(* PLC project mtcs_tmc, Institute of Astronomy Onto 0.0.1 *)
(* stored: creationDateTime 2025-05-06T14:59:44.773808, modificationDateTime 2025-05-06T14:59:44.773808 *)

TYPE TmcTimingMode : (LOCAL_CLOCK := 0, PTP_IEEE_1588 := 1);
END_TYPE

TYPE TmcAxesErrors : (AXES_NO_ERROR := 0, AXES_OBJECT_RC_OUT_OF_RANGE := 1, AXES_OBJECT_DC_OUT_OF_RANGE := 2, AXES_OBJECT_PR_OUT_OF_RANGE := 3, AXES_OBJECT_PD_OUT_OF_RANGE := 4, AXES_OBJECT_PX_OUT_OF_RANGE := 5, AXES_EQ_OUT_OF_RANGE := 6, AXES_LOCATION_XP_OUT_OF_RANGE := 7, AXES_LOCATION_YP_OUT_OF_RANGE := 8, AXES_LOCATION_DX_OUT_OF_RANGE := 9, AXES_LOCATION_DY_OUT_OF_RANGE := 10, AXES_LOCATION_ELONG_OUT_OF_RANGE := 11, AXES_LOCATION_PHI_OUT_OF_RANGE := 12, AXES_LOCATION_HM_OUT_OF_RANGE := 13, AXES_LOCATION_TK_OUT_OF_RANGE := 14, AXES_LOCATION_PHPA_OUT_OF_RANGE := 15, AXES_LOCATION_RH_OUT_OF_RANGE := 16, AXES_LOCATION_WLFQ_OUT_OF_RANGE := 17, AXES_LOCATION_TLR_OUT_OF_RANGE := 18, AXES_FEEDBACK_AZ_OUT_OF_RANGE := 19, AXES_FEEDBACK_EL_OUT_OF_RANGE := 20);
END_TYPE

TYPE TmcTimingErrors : (TIMING_NO_ERROR := 0, TIMING_DUT_OUT_OF_RANGE := 1, TIMING_GETCURDCTIME_FAILED := 2);
END_TYPE

TYPE TmcTarget : STRUCT
  {attribute 'TcHmiSymbol.Show'}
  rc : LREAL;  (* Object mean right ascention (alpha) in radians *)
  {attribute 'TcHmiSymbol.Show'}
  dc : LREAL;  (* Object mean declination (delta) in radians *)
  {attribute 'TcHmiSymbol.Show'}
  pr : INT;  (* Object Right Ascention proper motion in radians/year (do not multiply by cos(dc)!) *)
  {attribute 'TcHmiSymbol.Show'}
  pd : INT;  (* Object declination proper motion in radians/year *)
  {attribute 'TcHmiSymbol.Show'}
  px : LREAL;  (* Object parallax in arcseconds *)
  {attribute 'TcHmiSymbol.Show'}
  rv : LREAL;  (* Object radial velocity in km/s *)
END_STRUCT;
END_TYPE

TYPE TmcLocation : STRUCT
  {attribute 'TcHmiSymbol.Show'}
  xp : REAL;  (* Earth polar motion x in radians *)
  {attribute 'TcHmiSymbol.Show'}
  yp : REAL;  (* Earth polar motion y in radians *)
  {attribute 'TcHmiSymbol.Show'}
  dx : REAL;  (* Nutation adjustment dX in radians *)
  {attribute 'TcHmiSymbol.Show'}
  dy : REAL;  (* Nutation adjustment dY in radians *)
  {attribute 'TcHmiSymbol.Show'}
  elong : LREAL;  (* East longitude in radians *)
  {attribute 'TcHmiSymbol.Show'}
  phi : LREAL;  (* latitude in radians *)
  {attribute 'TcHmiSymbol.Show'}
  hm : REAL;  (* Height above sea level in meters *)
  {attribute 'TcHmiSymbol.Show'}
  tk : REAL;  (* Local temperature in Kelvin *)
  {attribute 'TcHmiSymbol.Show'}
  phpa : REAL;  (* Local pressure in hectoPascal = millibar *)
  {attribute 'TcHmiSymbol.Show'}
  rh : REAL;  (* Local relative humidity as a fraction (0...1) *)
  {attribute 'TcHmiSymbol.Show'}
  wlfq : REAL;  (* Observing wavelength in microns *)
  {attribute 'TcHmiSymbol.Show'}
  tlr : REAL;  (* Tropospheric lapse rate in K/m *)
END_STRUCT;
END_TYPE

TYPE TmcAzEl : STRUCT
  {attribute 'TcHmiSymbol.Show'}
  az : LREAL;  (* Azimuth in radians *)
  {attribute 'TcHmiSymbol.Show'}
  el : LREAL;  (* Elevation in radians *)
END_STRUCT;
END_TYPE

TYPE TmcAzElFull : STRUCT
  {attribute 'TcHmiSymbol.Show'}
  az : LREAL;  (* Azimuth in radians *)
  {attribute 'TcHmiSymbol.Show'}
  azd : LREAL;  (* Azimuth velocity in radians per second *)
  {attribute 'TcHmiSymbol.Show'}
  azdd : LREAL;  (* Azimuth acceleration in radians/s2 *)
  {attribute 'TcHmiSymbol.Show'}
  el : LREAL;  (* Elevation in radians *)
  {attribute 'TcHmiSymbol.Show'}
  eld : LREAL;  (* Elevation velocity in radians per second *)
  {attribute 'TcHmiSymbol.Show'}
  eldd : LREAL;  (* Elevation acceleration in radians/s2 *)
  {attribute 'TcHmiSymbol.Show'}
  pa : LREAL;  (* Parallactic Angle in radians *)
  {attribute 'TcHmiSymbol.Show'}
  pad : LREAL;  (* Parallactic Angle velocity in radians per second *)
  {attribute 'TcHmiSymbol.Show'}
  padd : LREAL;  (* Parallactic Angle acceleration in radians/s2 *)
END_STRUCT;
END_TYPE

TYPE TmcRaDec : STRUCT
  {attribute 'TcHmiSymbol.Show'}
  ra : LREAL;  (* Right ascention (alpha) in radians *)
  {attribute 'TcHmiSymbol.Show'}
  dec : LREAL;  (* Declination (delta) in radians *)
END_STRUCT;
END_TYPE

TYPE TmcObserved : STRUCT
  {attribute 'TcHmiSymbol.Show'}
  aob : LREAL;  (* Observed azimuth (radians: North=0, East=PI/2) *)
  {attribute 'TcHmiSymbol.Show'}
  zob : LREAL;  (* Observed zentih distance (radians) *)
  {attribute 'TcHmiSymbol.Show'}
  hob : LREAL;  (* Observed hour angle (radians) *)
  {attribute 'TcHmiSymbol.Show'}
  dob : LREAL;  (* Observed declination (radians) *)
  {attribute 'TcHmiSymbol.Show'}
  rob : LREAL;  (* Observed right ascention (radians) *)
END_STRUCT;
END_TYPE

TYPE TmcTrue : STRUCT
  {attribute 'TcHmiSymbol.Show'}
  elong : LREAL;  (* True longitude of the site (radians, east +ve) *)
  {attribute 'TcHmiSymbol.Show'}
  phi : LREAL;  (* True geodetic latitude of the site (radians) *)
  {attribute 'TcHmiSymbol.Show'}
  daz : LREAL;  (* Azimuth correction for true longitude and latitude (terrestrial - celestial, radians) *)
END_STRUCT;
END_TYPE

TYPE TmcProcessedTarget : STRUCT
  {attribute 'TcHmiSymbol.Show'}
  given : TmcTarget;  (* The originally given target *)
  {attribute 'TcHmiSymbol.Show'}
  apparent : TmcRaDec;  (* Apparent target position *)
  {attribute 'TcHmiSymbol.Show'}
  quick : TmcAzElFull;  (* Quick computation results of target (without atmospheric refraction) *)
  {attribute 'TcHmiSymbol.Show'}
  observed : TmcObserved;  (* Observed target position *)
  {attribute 'TcHmiSymbol.Show'}
  observedFull : TmcAzElFull;  (* Observed target position/velocity/acceleration *)
  {attribute 'TcHmiSymbol.Show'}
  isValid : BOOL;  (* Is the target valid? *)
  {attribute 'TcHmiSymbol.Show'}
  isTooLow : BOOL;  (* Is the target too low? *)
END_STRUCT;
END_TYPE

TYPE TmcProcessedFeedback : STRUCT
  {attribute 'TcHmiSymbol.Show'}
  apparent : TmcRaDec;  (* Apparent feedback position *)
  {attribute 'TcHmiSymbol.Show'}
  mean : TmcRaDec;  (* Mean feedback position *)
  {attribute 'TcHmiSymbol.Show'}
  isValid : BOOL;  (* Is the feedback valid? *)
  {attribute 'TcHmiSymbol.Show'}
  isTooLow : BOOL;  (* Is the feedback too low? *)
END_STRUCT;
END_TYPE

TYPE TmcDateTime : STRUCT
  {attribute 'TcHmiSymbol.Show'}
  years : DINT;  (* Years, e.g. 2016 *)
  {attribute 'TcHmiSymbol.Show'}
  months : DINT;  (* Months, [1..12] *)
  {attribute 'TcHmiSymbol.Show'}
  days : DINT;  (* Days, [1..31] *)
  {attribute 'TcHmiSymbol.Show'}
  hours : DINT;  (* Hours, [0..23] *)
  {attribute 'TcHmiSymbol.Show'}
  minutes : DINT;  (* Minutes, [0..59] *)
  {attribute 'TcHmiSymbol.Show'}
  seconds : DINT;  (* Secconds, [0..60] (60 during leap second event!) *)
  {attribute 'TcHmiSymbol.Show'}
  microseconds : DINT;  (* Microseconds, [0..999999] *)
  {attribute 'TcHmiSymbol.Show'}
  fractionOfDay : LREAL;  (* Fraction of the day, [0.0..1.0[ *)
END_STRUCT;
END_TYPE

TYPE TmcUnixTime : STRUCT
  {attribute 'TcHmiSymbol.Show'}
  sec : LINT;  (* Seconds from Jan 1, 1970 *)
  {attribute 'TcHmiSymbol.Show'}
  usec : LINT;  (* Microseconds *)
END_STRUCT;
END_TYPE

TYPE TmcUtcTime : STRUCT
  {attribute 'TcHmiSymbol.Show'}
  dcTime : LINT;  (* DC time *)
  {attribute 'TcHmiSymbol.Show'}
  mode : TmcTimingMode;  (* Local clock or PTP? *)
  {attribute 'TcHmiSymbol.Show'}
  unixTime : TmcUnixTime;  (* UTC as Unix time *)
  {attribute 'TcHmiSymbol.Show'}
  mjd : LREAL;  (* UTC as Modified Julian Days *)
  {attribute 'TcHmiSymbol.Show'}
  dateTime : TmcDateTime;  (* EtherCAT master: Offset between DC and TwinCAT time (in ns) *)
END_STRUCT;
END_TYPE

TYPE TmcUt1Time : STRUCT
  {attribute 'TcHmiSymbol.Show'}
  mjd : LREAL;  (* UT1 as Modified Julian Days *)
END_STRUCT;
END_TYPE

TYPE TmcFromIoEcatMaster : STRUCT
  {attribute 'TcHmiSymbol.Show'}
  dcToTcTimeOffset : LINT;  (* EtherCAT master: Offset between DC and TwinCAT time (in ns) *)
  {attribute 'TcHmiSymbol.Show'}
  dcToExtTimeOffset : LINT;  (* EtherCAT master: Offset between Dc and external time (in ns) *)
END_STRUCT;
END_TYPE

TYPE TmcFromIoEL6688 : STRUCT
  {attribute 'TcHmiSymbol.Show'}
  internalTimestamp : ULINT;  (* EL6688 module: internal timestamp *)
  {attribute 'TcHmiSymbol.Show'}
  externalTimestamp : ULINT;  (* EL6688 module: external timestamp *)
  {attribute 'TcHmiSymbol.Show'}
  notConnected : BOOL;  (* EL6688 module: not connected *)
  {attribute 'TcHmiSymbol.Show'}
  updateToggle : BOOL;  (* EL6688 module: update toggle *)
END_STRUCT;
END_TYPE

TYPE TmcFromIo : STRUCT
  {attribute 'TcHmiSymbol.Show'}
  fromEL6688 : TmcFromIoEL6688;  (* Connect to inputs of EL6688 *)
  {attribute 'TcHmiSymbol.Show'}
  fromEcatMaster : TmcFromIoEcatMaster;  (* Connect to inputs of EtherCAT master *)
END_STRUCT;
END_TYPE

TYPE TmcFromPlcAxes : STRUCT
  {attribute 'TcHmiSymbol.Show'}
  object : TmcTarget;  (* Target *)
  {attribute 'TcHmiSymbol.Show'}
  equinox : LREAL;  (* Epoch of mean equinoxes (e.g. 2000.0) *)
  {attribute 'TcHmiSymbol.Show'}
  location : TmcLocation;  (* Location of the observatory *)
  {attribute 'TcHmiSymbol.Show'}
  feedback : TmcAzEl;  (* Feedback position (by the encoders) *)
END_STRUCT;
END_TYPE

TYPE TmcFromPlcTiming : STRUCT
  {attribute 'TcHmiSymbol.Show'}
  dut : LREAL;  (* Delta UT (=UT1 - UTC, floating point between 0 and 1 second) *)
  {attribute 'TcHmiSymbol.Show'}
  leapSeconds : DINT;  (* Number of leap seconds *)
  {attribute 'TcHmiSymbol.Show'}
  alwaysUseLocalClock : BOOL;  (* If TRUE, then the local clock (source=LOCAL_CLOCK) will be used even if an external (more accurate!) clock is available *)
END_STRUCT;
END_TYPE

TYPE TmcFromPlc : STRUCT
  {attribute 'TcHmiSymbol.Show'}
  fromAxes : TmcFromPlcAxes;  (* Connect to outputs of PLC - MTCS - Axes *)
  {attribute 'TcHmiSymbol.Show'}
  fromTiming : TmcFromPlcTiming;  (* Connect to outputs of PLC - MTCS - Services/Timing *)
END_STRUCT;
END_TYPE

TYPE TmcToPlcAxes : STRUCT
  {attribute 'TcHmiSymbol.Show'}
  polmo : TmcTrue;  (* True longitude/latitude/azimuth after polar motion correction *)
  {attribute 'TcHmiSymbol.Show'}
  last : LREAL;  (* Local apparent sidereal time *)
  {attribute 'TcHmiSymbol.Show'}
  ha : LREAL;  (* Hour angle in radians *)
  {attribute 'TcHmiSymbol.Show'}
  object : TmcProcessedTarget;  (* Processed target *)
  {attribute 'TcHmiSymbol.Show'}
  feedback : TmcProcessedFeedback;  (* Processed feedback *)
  {attribute 'TcHmiSymbol.Show'}
  error : TmcAxesErrors;  (* 0 = no error *)
END_STRUCT;
END_TYPE

TYPE TmcToPlcTiming : STRUCT
  {attribute 'TcHmiSymbol.Show'}
  utc : TmcUtcTime;  (* UTC time *)
  {attribute 'TcHmiSymbol.Show'}
  ut1 : TmcUt1Time;  (* UT1 time *)
  {attribute 'TcHmiSymbol.Show'}
  error : TmcTimingErrors;  (* 0 = no error *)
END_STRUCT;
END_TYPE

TYPE TmcToPlc : STRUCT
  {attribute 'TcHmiSymbol.Show'}
  toAxes : TmcToPlcAxes;  (* Connect to inputs of PLC - MTCS - Axes *)
  {attribute 'TcHmiSymbol.Show'}
  toTiming : TmcToPlcTiming;  (* Connect to inputs of PLC - MTCS - Services/Timing *)
END_STRUCT;
END_TYPE
